(* Logix 5000 project; controller YST_Emu Emulate 5570 rev 31.11; software revision 31.00 *)

TASK _1Second (periodic, rate 1000 ms, priority 10, watchdog 500 ms) : _1Second
TASK MainTask (continuous, watchdog 500 ms) : MainProgram, First_Task

MODULES
   Local : Emulate 5570 (ICP 2, rev 31.11)
END_MODULES

TYPE CHECKWORD_FLAGS :   // Checkword Flags
STRUCT
   AUTODRV : DINT;   // Auto-Drive Bit No.
   CLOSEDFB : DINT;   // Closed Feedback Bit No.
   OPENFB : DINT;   // Open Feedback Bit No.
   OUTPUT : DINT;   // Output Bit No.
   MANDRV : DINT;   // Manual Drive Bit No.
   MANUAL : DINT;   // Manual Control Bit No.
   CHECKOFF : DINT;   // Checking Off Bit No.
   TRIPPED : DINT;   // Tripped Bit No.
   FAULT : DINT;   // Fault Bit No.
   SIMFAIL : DINT;   // Simulate Failure Bit
   PREVSCAN : DINT;   // Previous Scan State
   FAULTLOGGED : DINT;   // Fault Logged Flag From Scada
   HIGHLIGHT : DINT;   // Highlight on Graphics
   RUNFB : DINT;   // Pump/Drive Run Feedback
   HEALTHYFB : DINT;   // Pump Healthy Feedback
   NOTTRIPPEDFB : DINT;   // Pump Not Tripped Feedback
   HEALTHYFAULTLOGGED : DINT;   // Pump Not Healthy Fault Logged
   TRIPPEDFAULTLOGGED : DINT;   // Pump Tripped Fault Logged
   INPUTSTATUS : DINT;   // Bit Number for Digital Input Status
   INPUTSTATUSDEBOUNCED : DINT;   // Bit Number For Debounced Input Status
   ANALOGSIMULATION : DINT;   // Bit Number For Analog Simulation Enabled, Used By FactoryTalk
END_STRUCT
END_TYPE

TYPE PlantItem :   // Plant Item
STRUCT
   CW : DINT;   // Checkword
   CheckTime : DINT;   // Check Time
   CheckTimer : DINT;   // Check Time Timer
   DebounceTime : DINT;   // Debounce Time
   DebounceTimer : DINT;   // Debounce Timer
   DriveBits : DINT;   // Item Automatic Drive Bits
   Scaled : REAL;   // Analogue Value Scaled For Input/Output
   RawInput : REAL;   // Raw Input Copied for display On Factory Talk
END_STRUCT
END_TYPE

VAR_GLOBAL   (* controller tags *)
   _1s_pulse : BOOL;
   Alarm_Reset : BOOL;
   Analog_Fault_No : DINT := 30001;
   Analog_Simulation_Enabled : BOOL;
   CWD : CHECKWORD_FLAGS := (CLOSEDFB := 4, OPENFB := 3, OUTPUT := 7, MANDRV := 5, MANUAL := 6, CHECKOFF := 8, FAULT := 15, SIMFAIL := 2, PREVSCAN := 1, FAULTLOGGED := 14, HIGHLIGHT := 9, RUNFB := 3, HEALTHYFB := 10, NOTTRIPPEDFB := 11, HEALTHYFAULTLOGGED := 16, TRIPPEDFAULTLOGGED := 17, INPUTSTATUSDEBOUNCED := 18, ANALOGSIMULATION := 12);
   Default_Check_Time : DINT;
   FV_B86 : INT[255];
        [0].1   // YST CIP Running
   FV_N139 : INT[255] := ([0] := 95, [1] := -32767, [2] := -32767, [3] := -32767, [4] := -32767, [5] := -32767, [6] := -32767, [7] := -32767, [8] := -32767, [9] := -32767, [10] := -32767, [11] := -32767, [12] := -32767, [13] := 32767, [14] := -32767, [15] := 20, [17] := -32767, [18] := -32767, [19] := -32767, [20] := 9785, [21] := -32767, [22] := 32767, [23] := 3, [24] := 10, [25] := 86, [26] := -32767, [27] := 9789, [29] := 257, [30] := 59);   // YST1
        [30].0   // YST1 cooling required
        [0]   // YST1 attemperation control data
        [30].1   // YST1 low level covered flag
   FV_N140 : INT[255] := ([0] := 96, [2] := 30, [3] := 400, [4] := 30, [5] := 800, [6] := 30, [7] := 1200, [8] := 30, [9] := 1600, [10] := 30, [11] := 2000, [12] := 30, [13] := 32767, [14] := 30, [15] := 20, [16] := -32767, [17] := -32767, [18] := -32767, [19] := -32767, [20] := -31070, [21] := -32767, [22] := -31070, [23] := 1, [25] := 52, [30] := 34);   // YST2
        [30].0   // YST2 cooling required
        [0]   // YST2 attemperation control data
        [30].1   // YST2 low level covered flag
   FV_N80 : INT[255] := ([1] := 1);
   FV_N81 : INT[255];
   FV_N84 : INT[255];   // YST CIP Selected YST
   FV_N85 : INT[255];   // YST CIP Process Step
   FV_R2V1 : PlantItem := (CheckTime := 4, CheckTimer := 4, DriveBits := 2);   // R2V1
   FV_R2V2 : PlantItem := (CheckTime := 4, CheckTimer := 4);   // R2V2
   FV_TTX_YS_001_AI : PlantItem;
   FV_WYTR1 : PlantItem := (CheckTime := 8, CheckTimer := 8, DriveBits := 1);   // WYTR1
   FV_WYTR2 : PlantItem := (CheckTime := 4, CheckTimer := 4);   // WYTR2
   FV_YST01_LTX501_AI : PlantItem := (CW := 49152, CheckTime := 10, CheckTimer := 10, Scaled := 31.25, RawInput := 6000.0);
   FV_YST01_LTX501_AI_RawInput : DINT := 6000;
   FV_YST01_LTX501_ALARM : ALARM_DIGITAL;
   FV_YST01_LTX501_Cool_Lvl_OK : TIMER := (PRE := 2500);
   FV_YST01_LTX501_Fill_Lvl_OK : TIMER := (PRE := 2500, ACC := 2519, EN := 1, DN := 1);
   FV_YST01_LTX501_Timer_HiLevel : TIMER;
   FV_YST02_LTX501_AI : PlantItem := (CW := 32768, Scaled := 15.625, RawInput := 5000.0);
   FV_YST02_LTX501_AI_RawInput : DINT := 5000;
   FV_YST02_LTX501_ALARM : ALARM_DIGITAL;
   FV_YST02_LTX501_Cool_Lvl_OK : TIMER := (PRE := 2500);
   FV_YST02_LTX501_Fill_Lvl_OK : TIMER := (PRE := 2500);
   FV_YST02_LTX501_Timer_HiLevel : TIMER := (PRE := 10000);
   FV_YSV1CV : PlantItem := (CheckTime := 8);   // YSV1CV
   FV_YSV2CV : PlantItem := (CheckTime := 8);   // YSV2CV
   ItoF_raw_input : INT := 5000;
   One_Second_One_Scan : BOOL;
   overrange_RIO_analog_value : DINT;
   scale_analog_result : REAL := 15.625;
   scale_eu_max : REAL := 250.0;
   scale_eu_min : REAL;
   scale_raw_input : REAL := 5000.0;
   scale_raw_max : REAL := 20000.0;
   scale_raw_min : REAL := 4000.0;
   scale_routine_active : BOOL := 1;
   scale_temp : REAL := 0.015625;
   underrange_RIO_analog_value : DINT;
END_VAR

PROGRAM _1Second

ROUTINE OneSecond   (* ladder *)
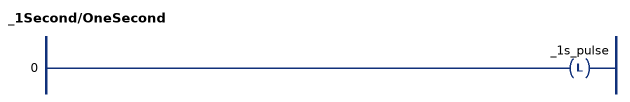
   0: OTL(_1s_pulse);
END_ROUTINE
END_PROGRAM

PROGRAM First_Task   (* main routine MainRoutine *)

ROUTINE MainRoutine   (* ladder *)
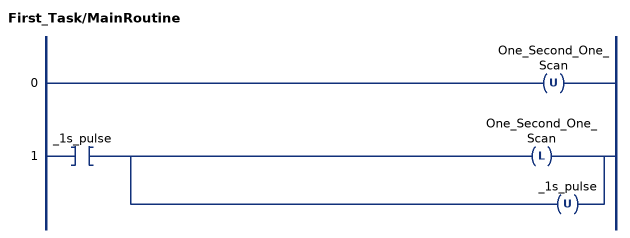
   0: OTU(One_Second_One_Scan);
   1: XIC(_1s_pulse)[OTL(One_Second_One_Scan) ,OTU(_1s_pulse) ];
END_ROUTINE
END_PROGRAM

PROGRAM MainProgram   (* main routine MainRoutine *)

ROUTINE Analog_Scale_ItoF   (* ladder *)
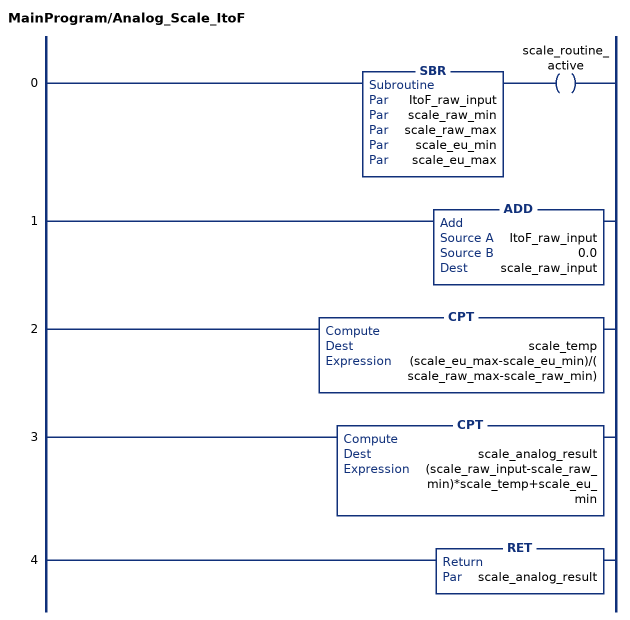
   0: SBR(ItoF_raw_input,scale_raw_min,scale_raw_max,scale_eu_min,scale_eu_max)OTE(scale_routine_active);
   1: ADD(ItoF_raw_input,0.0,scale_raw_input);
   2: CPT(scale_temp,(scale_eu_max-scale_eu_min)/(scale_raw_max-scale_raw_min));
   3: CPT(scale_analog_result,(scale_raw_input-scale_raw_min)*scale_temp+scale_eu_min);
   4: RET(scale_analog_result);
END_ROUTINE

ROUTINE FV_Analogs   (* ladder *)
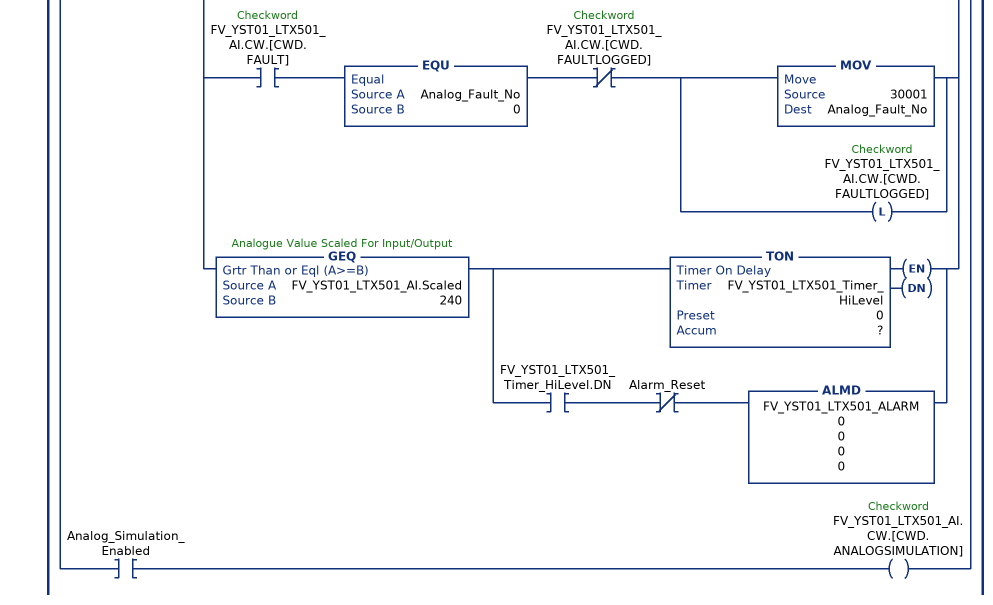
   0: [XIO(Analog_Simulation_Enabled) [XIO(FV_YST01_LTX501_AI.CW.[CWD.MANUAL]) JSR(Analog_Scale_ItoF,5,FV_YST01_LTX501_AI_RawInput,4000.0,20000.0,0.0,250.0,FV_YST01_LTX501_AI.Scaled) ,MOV(FV_YST01_LTX501_AI_RawInput,FV_YST01_LTX501_AI.RawInput) ,[LIM(underrange_RIO_analog_value,FV_YST01_LTX501_AI_RawInput,overrange_RIO_analog_value) ,XIC(FV_YST01_LTX501_AI.CW.[CWD.CHECKOFF]) ] CLR(FV_YST01_LTX501_AI.CheckTimer) ,XIC(S:FS) [OTU(FV_YST01_LTX501_AI.CW.[CWD.MANUAL]) ,LEQ(FV_YST01_LTX501_AI.CheckTime,0) MOV(Default_Check_Time,FV_YST01_LTX501_AI.CheckTime) ] ,XIC(One_Second_One_Scan) LES(FV_YST01_LTX501_AI.CheckTimer,FV_YST01_LTX501_AI.CheckTime) ADD(FV_YST01_LTX501_AI.CheckTimer,1,FV_YST01_LTX501_AI.CheckTimer) ,GEQ(FV_YST01_LTX501_AI.CheckTimer,FV_YST01_LTX501_AI.CheckTime) XIO(Alarm_Reset) OTE(FV_YST01_LTX501_AI.CW.[CWD.FAULT]) ,XIC(FV_YST01_LTX501_AI.CW.[CWD.FAULT]) EQU(Analog_Fault_No,0) XIO(FV_YST01_LTX501_AI.CW.[CWD.FAULTLOGGED]) [MOV(30001,Analog_Fault_No) ,OTL(FV_YST01_LTX501_AI.CW.[CWD.FAULTLOGGED]) ] ,GEQ(FV_YST01_LTX501_AI.Scaled,240) [TON(FV_YST01_LTX501_Timer_HiLevel,?,?) ,XIC(FV_YST01_LTX501_Timer_HiLevel.DN) XIO(Alarm_Reset) ALMD(FV_YST01_LTX501_ALARM,0,0,0,0) ] ] ,XIC(Analog_Simulation_Enabled) OTE(FV_YST01_LTX501_AI.CW.[CWD.ANALOGSIMULATION]) ];
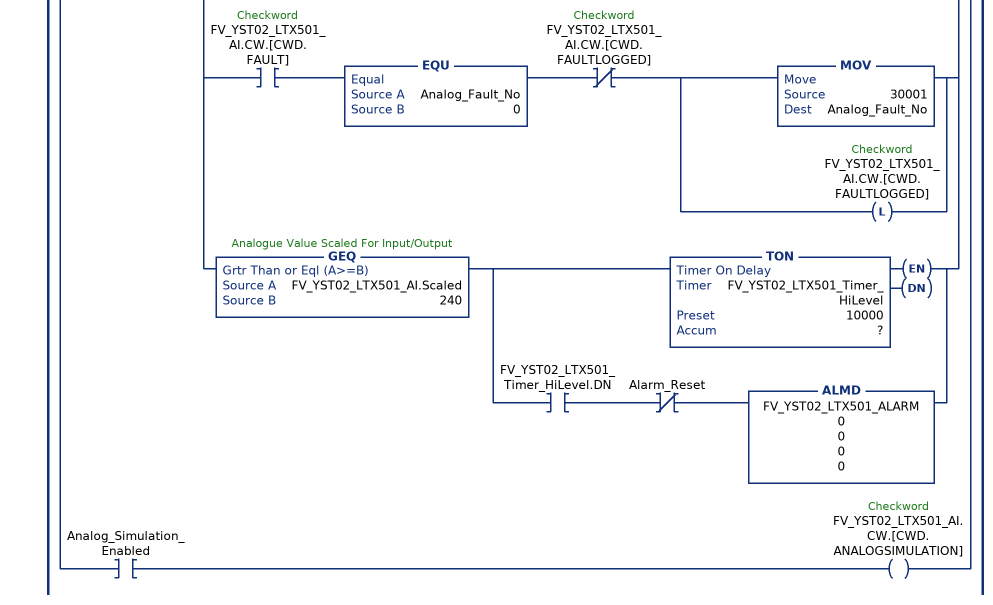
   1: [XIO(Analog_Simulation_Enabled) [XIO(FV_YST02_LTX501_AI.CW.[CWD.MANUAL]) JSR(Analog_Scale_ItoF,5,FV_YST02_LTX501_AI_RawInput,4000.0,20000.0,0.0,250.0,FV_YST02_LTX501_AI.Scaled) ,MOV(FV_YST02_LTX501_AI_RawInput,FV_YST02_LTX501_AI.RawInput) ,[LIM(underrange_RIO_analog_value,FV_YST02_LTX501_AI_RawInput,overrange_RIO_analog_value) ,XIC(FV_YST02_LTX501_AI.CW.[CWD.CHECKOFF]) ] CLR(FV_YST02_LTX501_AI.CheckTimer) ,XIC(S:FS) [OTU(FV_YST02_LTX501_AI.CW.[CWD.MANUAL]) ,LEQ(FV_YST02_LTX501_AI.CheckTime,0) MOV(Default_Check_Time,FV_YST02_LTX501_AI.CheckTime) ] ,XIC(One_Second_One_Scan) LES(FV_YST02_LTX501_AI.CheckTimer,FV_YST02_LTX501_AI.CheckTime) ADD(FV_YST02_LTX501_AI.CheckTimer,1,FV_YST02_LTX501_AI.CheckTimer) ,GEQ(FV_YST02_LTX501_AI.CheckTimer,FV_YST02_LTX501_AI.CheckTime) XIO(Alarm_Reset) OTE(FV_YST02_LTX501_AI.CW.[CWD.FAULT]) ,XIC(FV_YST02_LTX501_AI.CW.[CWD.FAULT]) EQU(Analog_Fault_No,0) XIO(FV_YST02_LTX501_AI.CW.[CWD.FAULTLOGGED]) [MOV(30001,Analog_Fault_No) ,OTL(FV_YST02_LTX501_AI.CW.[CWD.FAULTLOGGED]) ] ,GEQ(FV_YST02_LTX501_AI.Scaled,240) [TON(FV_YST02_LTX501_Timer_HiLevel,?,?) ,XIC(FV_YST02_LTX501_Timer_HiLevel.DN) XIO(Alarm_Reset) ALMD(FV_YST02_LTX501_ALARM,0,0,0,0) ] ] ,XIC(Analog_Simulation_Enabled) OTE(FV_YST02_LTX501_AI.CW.[CWD.ANALOGSIMULATION]) ];
END_ROUTINE

ROUTINE FV_FV_VALVES_105   (* ladder *)
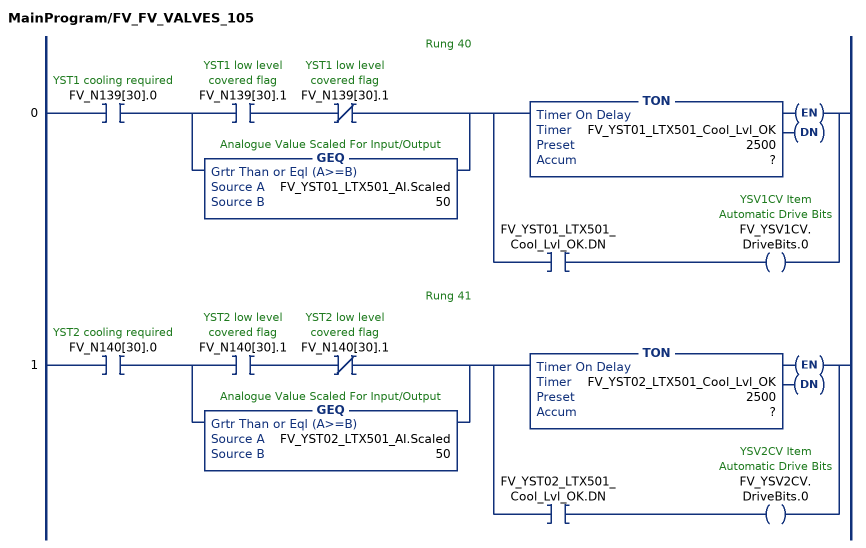
   // Rung 40
   0: XIC(FV_N139[30].0)[XIC(FV_N139[30].1) XIO(FV_N139[30].1) ,GEQ(FV_YST01_LTX501_AI.Scaled,50) ][TON(FV_YST01_LTX501_Cool_Lvl_OK,?,?) ,XIC(FV_YST01_LTX501_Cool_Lvl_OK.DN) OTE(FV_YSV1CV.DriveBits.0) ];
   // Rung 41
   1: XIC(FV_N140[30].0)[XIC(FV_N140[30].1) XIO(FV_N140[30].1) ,GEQ(FV_YST02_LTX501_AI.Scaled,50) ][TON(FV_YST02_LTX501_Cool_Lvl_OK,?,?) ,XIC(FV_YST02_LTX501_Cool_Lvl_OK.DN) OTE(FV_YSV2CV.DriveBits.0) ];
END_ROUTINE

ROUTINE FV_YSTFILL_PR_82   (* ladder *)
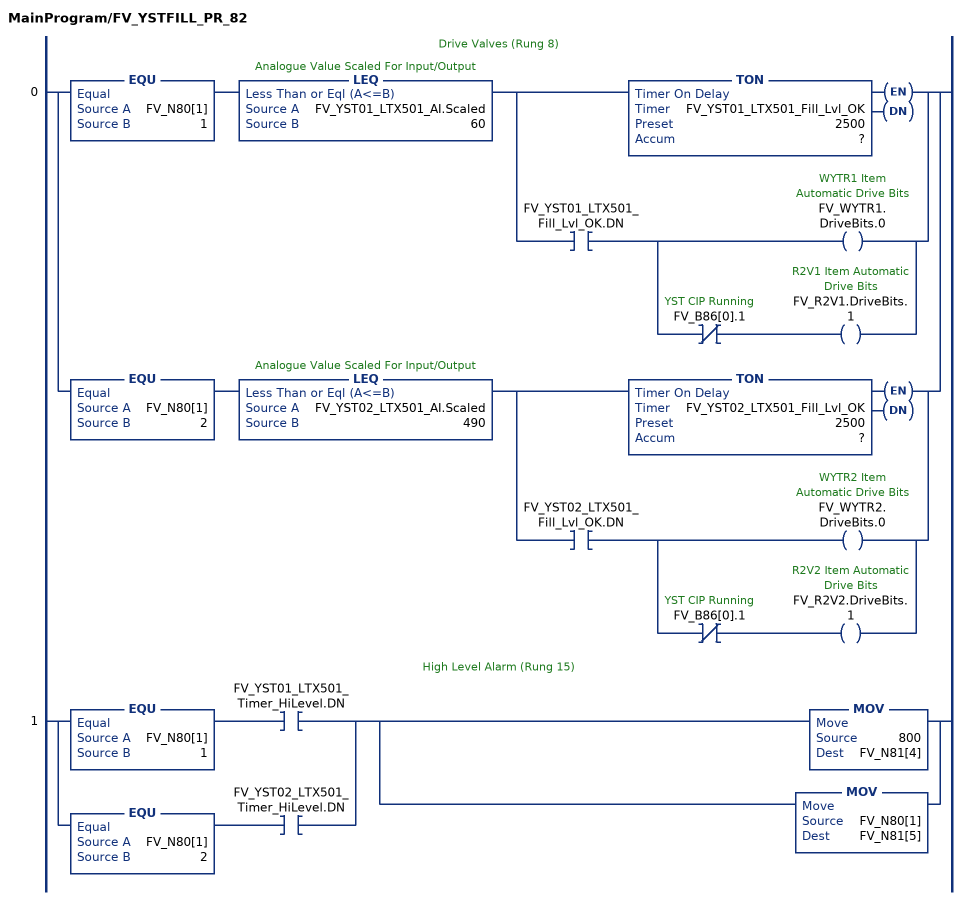
   // Drive Valves (Rung 8)
   0: [EQU(FV_N80[1],1) LEQ(FV_YST01_LTX501_AI.Scaled,60) [TON(FV_YST01_LTX501_Fill_Lvl_OK,?,?) ,XIC(FV_YST01_LTX501_Fill_Lvl_OK.DN) [OTE(FV_WYTR1.DriveBits.0) ,XIO(FV_B86[0].1) OTE(FV_R2V1.DriveBits.1) ] ] ,EQU(FV_N80[1],2) LEQ(FV_YST02_LTX501_AI.Scaled,490) [TON(FV_YST02_LTX501_Fill_Lvl_OK,?,?) ,XIC(FV_YST02_LTX501_Fill_Lvl_OK.DN) [OTE(FV_WYTR2.DriveBits.0) ,XIO(FV_B86[0].1) OTE(FV_R2V2.DriveBits.1) ] ] ];
   // High Level Alarm (Rung 15)
   1: [EQU(FV_N80[1],1) XIC(FV_YST01_LTX501_Timer_HiLevel.DN) ,EQU(FV_N80[1],2) XIC(FV_YST02_LTX501_Timer_HiLevel.DN) ][MOV(800,FV_N81[4]) ,MOV(FV_N80[1],FV_N81[5]) ];
END_ROUTINE

ROUTINE MainRoutine   (* ladder *)
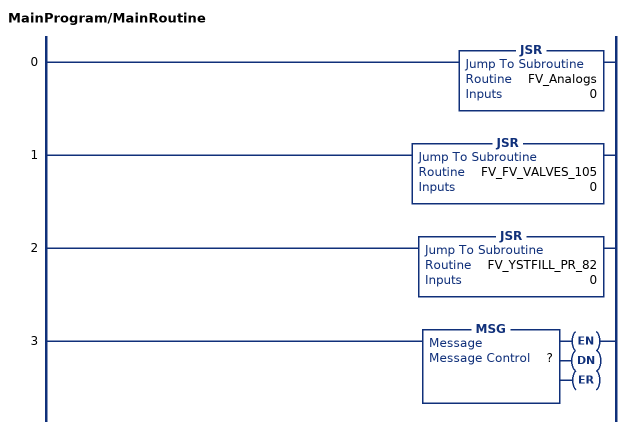
   0: JSR(FV_Analogs,0);
   1: JSR(FV_FV_VALVES_105,0);
   2: JSR(FV_YSTFILL_PR_82,0);
   3 (stored rung type 13): MSG(?);
END_ROUTINE
END_PROGRAM
